// TIA Portal V17 export
// export: Created 2022-03-12T16:05:13.5325441Z, ExportSetting WithDefaults, DisplayName Totally Integrated Automation Portal, DisplayVersion V17, DisplayName TIA Portal Openness, DisplayVersion V17, DisplayName TIA Portal Version Control Interface, DisplayVersion V17, DisplayName STEP 7 Professional, DisplayVersion V17, DisplayName STEP 7 Safety, DisplayVersion V17, DisplayName WinCC Advanced / Unified PC, DisplayVersion V17
FUNCTION_BLOCK "UN_00_Main"   // FB31620, LAD
TITLE = UN_00_Main
{ S7_Optimized_Access := 'TRUE' }
AUTHOR : tech.team.motioncontrol@siemens.com
FAMILY : CPG
VERSION : 1.0
// Support: tech.team.motioncontrol@siemens.com
// Fax: +49 (0) 9131/98-1297
// stored: AutoNumber true, IsIECCheckEnabled false, IsRetainMemResEnabled false, MemoryReserve 100, SetENOAutomatically false, UDAEnableTagReadback false
   VAR
      instPackML_ModuleSum { ExternalAccessible := 'False'; ExternalVisible := 'False'; ExternalWritable := 'False'; S7_SetPoint := 'True'} : "UN_01_PackML_ModuleSum";   // PackML Module Summation Logic of EM-level command and state complete's to unit level
      instPackML { ExternalAccessible := 'False'; ExternalVisible := 'False'; ExternalWritable := 'False'; S7_SetPoint := 'True'} : "UN_02_PackML";
      instLineComm { ExternalAccessible := 'False'; ExternalVisible := 'False'; ExternalWritable := 'False'; S7_SetPoint := 'True'} : "UN_03_LineComm";
      instEventControl { ExternalAccessible := 'False'; ExternalVisible := 'False'; ExternalWritable := 'False'; S7_SetPoint := 'True'} : "UN_04_EventControl";
      instEventSummation { ExternalAccessible := 'False'; ExternalVisible := 'False'; ExternalWritable := 'False'; S7_SetPoint := 'True'} : "UN_05_EventSummation";
      instMiscFunctions { ExternalAccessible := 'False'; ExternalVisible := 'False'; ExternalWritable := 'False'; S7_SetPoint := 'True'} : "UN_06_MiscFunctions";
      instRecipeControl { ExternalAccessible := 'False'; ExternalVisible := 'False'; ExternalWritable := 'False'; S7_SetPoint := 'True'} : "UN_07_RecipeControl";
   END_VAR
   VAR_TEMP   // added for the SCL form of the ladder/FBD networks
      _w1 : Bool;
   END_VAR
BEGIN

REGION Network 1: Call the PackML Module Summation Logic
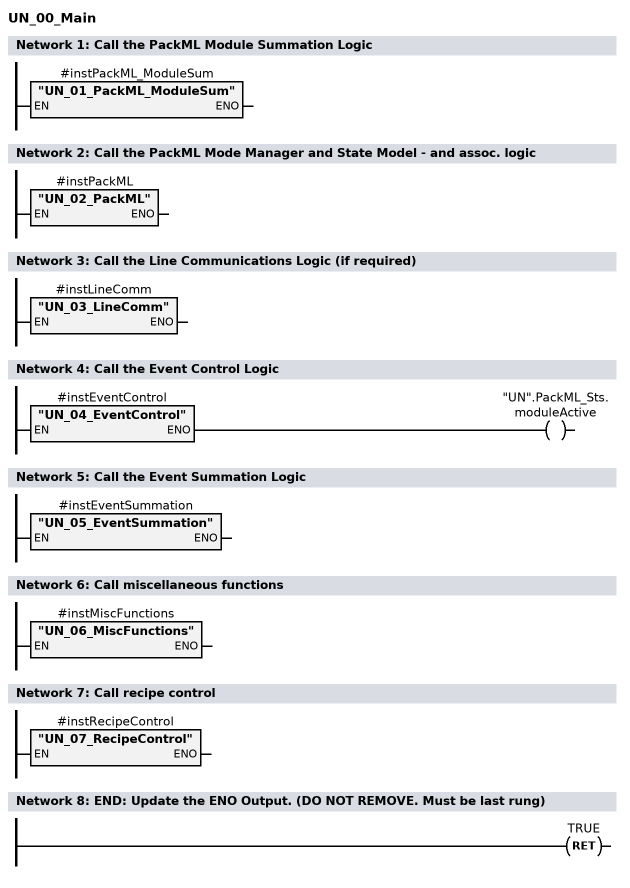
   RUNG wire#powerrail
      #instPackML_ModuleSum()
   END_RUNG
   // the same network as SCL:
   #instPackML_ModuleSum();   // "UN_01_PackML_ModuleSum"
END_REGION

REGION Network 2: Call the PackML Mode Manager and State Model - and assoc. logic
   RUNG wire#powerrail
      #instPackML()
   END_RUNG
   // the same network as SCL:
   #instPackML();   // "UN_02_PackML"
END_REGION

REGION Network 3: Call the Line Communications Logic (if required)
   RUNG wire#powerrail
      #instLineComm()
   END_RUNG
   // the same network as SCL:
   #instLineComm();   // "UN_03_LineComm"
END_REGION

REGION Network 4: Call the Event Control Logic
   RUNG wire#powerrail
      #instEventControl()
      Coil( "UN".PackML_Sts.moduleActive )
   END_RUNG
   // the same network as SCL:
   #instEventControl(ENO => #_w1);   // "UN_04_EventControl"
   "UN".PackML_Sts.moduleActive := #_w1;
END_REGION

REGION Network 5: Call the Event Summation Logic
   RUNG wire#powerrail
      #instEventSummation()
   END_RUNG
   // the same network as SCL:
   #instEventSummation();   // "UN_05_EventSummation"
END_REGION

REGION Network 6: Call miscellaneous functions
   RUNG wire#powerrail
      #instMiscFunctions()
   END_RUNG
   // the same network as SCL:
   #instMiscFunctions();   // "UN_06_MiscFunctions"
END_REGION

REGION Network 7: Call recipe control
   RUNG wire#powerrail
      #instRecipeControl()
   END_RUNG
   // the same network as SCL:
   #instRecipeControl();   // "UN_07_RecipeControl"
END_REGION

REGION Network 8: END: Update the ENO Output. (DO NOT REMOVE. Must be last rung)
   RUNG wire#powerrail
      ReturnCoil( TRUE )
   END_RUNG
   // the same network as SCL:
   ENO := TRUE;
   RETURN;
END_REGION
END_FUNCTION_BLOCK
